FUNCTION_BLOCK BaseXmlDataSrvProcess EXTENDS SM_BaseMcProcess
VAR_INPUT
END_VAR
VAR_OUTPUT
END_VAR
VAR
	testVar3 : BOOL;
END_VAR

SUPER^();

END_FUNCTION_BLOCK

(* stored: Version 1.1.0.1, ProductVersion 3.1.4018.2
   POU BaseXmlDataSrvProcess: Id {512d9e18-f729-4408-b671-547062c42270}, SpecialFunc None *)
